FUNCTION_BLOCK Mode (* Composite Function Block Type *)
  (* Standard: 61499-2 *)
  (* Version 0.0, 19/05/2022, SESA371406, Schneider Electric, template *)
  PACKAGE SE.Nereda;
  {SET_ATTRIBUTE(CompilerOptions, CheckConnectionsStrictly=False)}
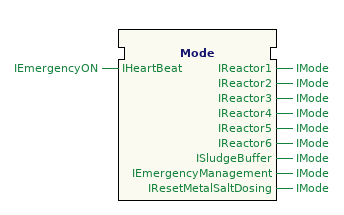
  SOCKETS
    IHeartBeat : IEmergencyON;
  END_SOCKETS
  PLUGS
    IReactor1 : IMode;
    IReactor2 : IMode;
    IReactor3 : IMode;
    IReactor4 : IMode;
    IReactor5 : IMode;
    IReactor6 : IMode;
    ISludgeBuffer : IMode;
    IEmergencyManagement : IMode;
    IResetMetalSaltDosing : IMode;
  END_PLUGS
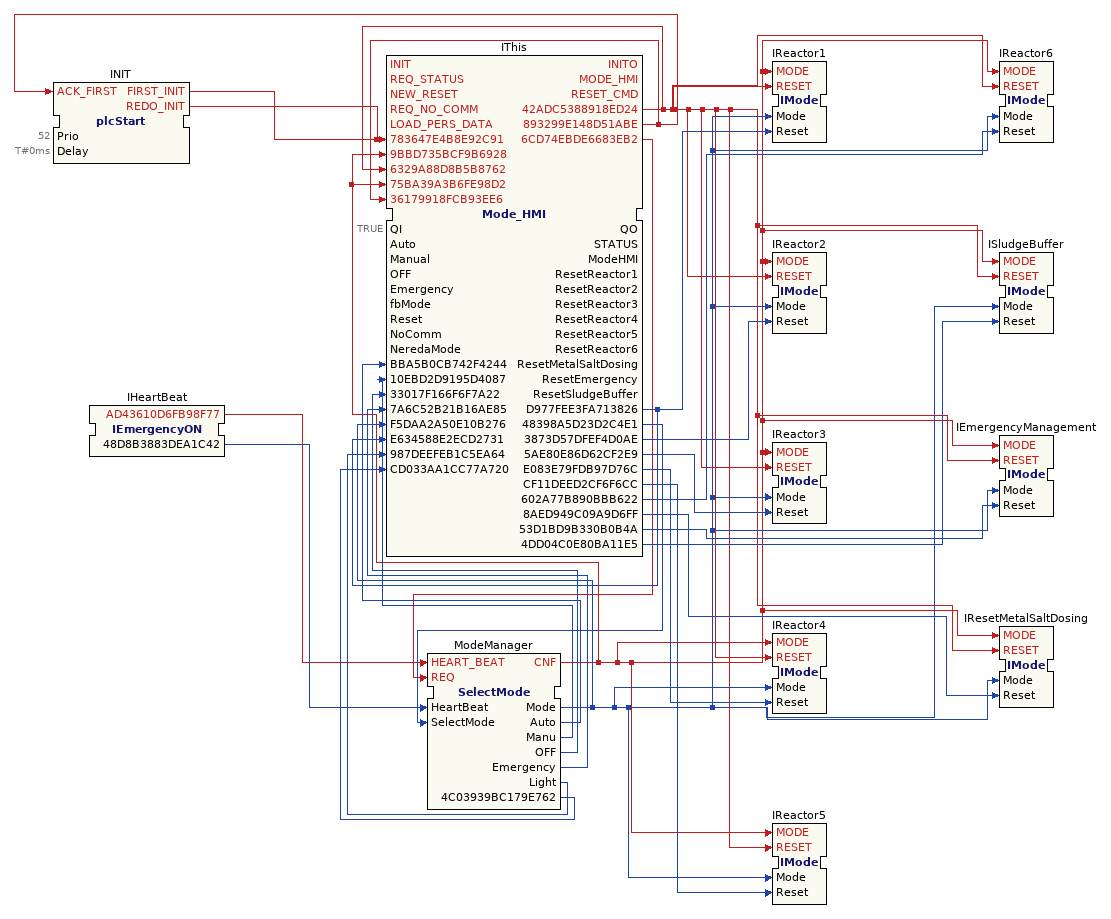
  (* 01 - FUNCTIONNAL INPUT INTERFACE *)
  (* 00 - INITIALIZATION *)
  (* 05 - LOGIC *)
  (* 06 - HMI INTERFACE *)
  (* 02 - FUNCTIONNAL OUTPUT INTERFACE *)
  (* Reactor Logic *)
  (* Mode : 0 : Automatic Mode 1 : Off 2 : Manual Mode 3 : Emergency Mode *)
  (* ModeNereda : 2 : Automatic Mode 0 : Off 1 : Manual Mode -1 : Emergency Mode *)
  FBS
    IThis : Mode_HMI(QI := TRUE);
    INIT : plcStart(Prio := 52, Delay := T#0ms);
    ModeManager : SelectMode;
  END_FBS
  EVENT_CONNECTIONS
    ModeManager.CNF TO IReactor1.MODE;
    ModeManager.CNF TO IReactor6.MODE;
    ModeManager.CNF TO IReactor2.MODE;
    ModeManager.CNF TO ISludgeBuffer.MODE;
    ModeManager.CNF TO IReactor3.MODE;
    ModeManager.CNF TO IEmergencyManagement.MODE;
    ModeManager.CNF TO IReactor4.MODE;
    ModeManager.CNF TO IResetMetalSaltDosing.MODE;
    ModeManager.CNF TO IReactor5.MODE;
    IHeartBeat.AD43610D6FB98F77 TO ModeManager.HEART_BEAT;
    INIT.FIRST_INIT TO IThis.783647E4B8E92C91;
    INIT.REDO_INIT TO IThis.783647E4B8E92C91;
    ModeManager.CNF TO IThis.9BBD735BCF9B6928;
    IThis.42ADC5388918ED24 TO IThis.6329A88D8B5B8762;
    ModeManager.CNF TO IThis.75BA39A3B6FE98D2;
    IThis.893299E148D51ABE TO IThis.36179918FCB93EE6;
    IThis.893299E148D51ABE TO INIT.ACK_FIRST;
    IThis.6CD74EBDE6683EB2 TO ModeManager.REQ;
    IThis.42ADC5388918ED24 TO IReactor1.RESET;
    IThis.42ADC5388918ED24 TO IReactor6.RESET;
    IThis.42ADC5388918ED24 TO IReactor2.RESET;
    IThis.42ADC5388918ED24 TO ISludgeBuffer.RESET;
    IThis.42ADC5388918ED24 TO IReactor3.RESET;
    IThis.42ADC5388918ED24 TO IEmergencyManagement.RESET;
    IThis.42ADC5388918ED24 TO IReactor4.RESET;
    IThis.42ADC5388918ED24 TO IResetMetalSaltDosing.RESET;
    IThis.42ADC5388918ED24 TO IReactor5.RESET;
  END_CONNECTIONS
  DATA_CONNECTIONS
    ModeManager.Mode TO IReactor1.Mode;
    ModeManager.Mode TO IReactor6.Mode;
    ModeManager.Mode TO IReactor2.Mode;
    ModeManager.Mode TO ISludgeBuffer.Mode;
    ModeManager.Mode TO IReactor3.Mode;
    ModeManager.Mode TO IEmergencyManagement.Mode;
    ModeManager.Mode TO IReactor4.Mode;
    ModeManager.Mode TO IResetMetalSaltDosing.Mode;
    ModeManager.Mode TO IReactor5.Mode;
    IHeartBeat.48D8B3883DEA1C42 TO ModeManager.HeartBeat;
    ModeManager.Auto TO IThis.BBA5B0CB742F4244;
    ModeManager.Manu TO IThis.10EBD2D9195D4087;
    ModeManager.OFF TO IThis.33017F166F6F7A22;
    ModeManager.Emergency TO IThis.7A6C52B21B16AE85;
    ModeManager.Mode TO IThis.F5DAA2A50E10B276;
    IThis.D977FEE3FA713826 TO IThis.E634588E2ECD2731;
    ModeManager.Light TO IThis.987DEEFEB1C5EA64;
    ModeManager.4C03939BC179E762 TO IThis.CD033AA1CC77A720;
    IThis.48398A5D23D2C4E1 TO ModeManager.SelectMode;
    IThis.D977FEE3FA713826 TO IReactor1.Reset;
    IThis.3873D57DFEF4D0AE TO IReactor2.Reset;
    IThis.5AE80E86D62CF2E9 TO IReactor3.Reset;
    IThis.E083E79FDB97D76C TO IReactor4.Reset;
    IThis.CF11DEED2CF6F6CC TO IReactor5.Reset;
    IThis.602A77B890BBB622 TO IReactor6.Reset;
    IThis.8AED949C09A9D6FF TO IResetMetalSaltDosing.Reset;
    IThis.53D1BD9B330B0B4A TO IEmergencyManagement.Reset;
    IThis.4DD04C0E80BA11E5 TO ISludgeBuffer.Reset;
  END_CONNECTIONS
END_FUNCTION_BLOCK
